// TIA Portal V15.1 export
// export: Created 2024-05-17T05:38:40.0003593Z, ExportSetting WithDefaults, DisplayName Totally Integrated Automation Portal, DisplayVersion V15.1 Update 5, DisplayName TIA Portal Openness, DisplayVersion V15.1 Update 5, DisplayName SINAMICS Startdrive Advanced, DisplayVersion V15.1, DisplayName G130, G150, S120, S150, SINAMICS MV, S210, DisplayVersion V15.1, DisplayName G110M, G120, G120C, G120D, G120P, DisplayVersion V15.1, DisplayName STEP 7 Professional, DisplayVersion V15.1 Update 5, DisplayName STEP 7 Safety, DisplayVersion V15.1, DisplayName WinCC Professional, DisplayVersion V15.1 Update 5, DisplayName SIMATIC Visualization Architect, DisplayVersion V15.1
FUNCTION_BLOCK "LGBProcessLighting"   // FB6697, FBD
TITLE = LGBProcessLighting
{ S7_Optimized_Access := 'TRUE' }
VERSION : 0.1
// stored: AutoNumber false, IsIECCheckEnabled false, IsRetainMemResEnabled false, MemoryReserve 100, SetENOAutomatically False, UDAEnableTagReadback false
   VAR_INPUT
      I_StartProduction { ExternalAccessible := 'False'; ExternalVisible := 'False'; ExternalWritable := 'False'} : Bool;   // Start Production line
      I_StopProduction { ExternalAccessible := 'False'; ExternalVisible := 'False'; ExternalWritable := 'False'} : Bool;   // Stop Production line
      I_StartReqCR { ExternalAccessible := 'False'; ExternalVisible := 'False'; ExternalWritable := 'False'} : Bool;   // Start request by controlroom
      I_StoppedByCR { ExternalAccessible := 'False'; ExternalVisible := 'False'; ExternalWritable := 'False'} : Bool;   // Production line stopped by control room
      I_BodyNumber { ExternalAccessible := 'False'; ExternalVisible := 'False'; ExternalWritable := 'False'} : DWord;   // Body number
      I_TopCoatColour { ExternalAccessible := 'False'; ExternalVisible := 'False'; ExternalWritable := 'False'} : Int;   // Top coat colour
      I_ColourGroup { ExternalAccessible := 'False'; ExternalVisible := 'False'; ExternalWritable := 'False'} : "ColourGroup";   // High speed value 0-100% / Colour Group
   END_VAR
   VAR_OUTPUT
      O_BreakMode { ExternalAccessible := 'False'; ExternalVisible := 'False'; ExternalWritable := 'False'} : Bool;   // Output 1 - Break Mode
      O_Intensity1 { ExternalAccessible := 'False'; ExternalVisible := 'False'; ExternalWritable := 'False'} : Bool;   // Output 2 - Intensity 1
      O_Intensity2 { ExternalAccessible := 'False'; ExternalVisible := 'False'; ExternalWritable := 'False'} : Bool;   // Output 3 - Intensity 2
      O_Intensity3 { ExternalAccessible := 'False'; ExternalVisible := 'False'; ExternalWritable := 'False'} : Bool;   // Output 4 - Intensity 3
      O_AlarmABCondition { ExternalAccessible := 'False'; ExternalVisible := 'False'; ExternalWritable := 'False'} : Bool;   // Alarm AB Condition
      O_AlarmA { ExternalAccessible := 'False'; ExternalVisible := 'False'; ExternalWritable := 'False'} : Bool;   // Alarm A
      O_AlarmB { ExternalAccessible := 'False'; ExternalVisible := 'False'; ExternalWritable := 'False'} : Bool;   // Alarm B
      O_AlarmC { ExternalAccessible := 'False'; ExternalVisible := 'False'; ExternalWritable := 'False'} : Bool;   // Alarm C
      O_AlarmD { ExternalAccessible := 'False'; ExternalVisible := 'False'; ExternalWritable := 'False'} : Bool;   // Alarm D
      H_AlarmDWord { ExternalAccessible := 'False'; ExternalVisible := 'False'; ExternalWritable := 'False'} : DWord;   // Alarm Word
   END_VAR
   VAR_IN_OUT
      H_HMI : "H_HMI";   // Icon Animation
      H_GBProcessLighting : "H_GBProcessLighting";   // Animation
      C_ProcessLightingConfig : "ProcessLightingConfig";   // Config
      IO_IDWorkStation { ExternalAccessible := 'False'; ExternalVisible := 'False'; ExternalWritable := 'False'} : Int;   // ID
      IO_GlobalOutput { ExternalAccessible := 'False'; ExternalVisible := 'False'; ExternalWritable := 'False'} : Bool;   // Global output
   END_VAR
   VAR
      AC_TopCoatColour { ExternalAccessible := 'False'; ExternalVisible := 'False'; ExternalWritable := 'False'} : Bool;   // Top Coat Colour is not configured in a colour group
      AD_ForceBreakMode { ExternalAccessible := 'False'; ExternalVisible := 'False'; ExternalWritable := 'False'} : Bool;   // Force process lighting active for Break Mode
      AD_ForceIntensity1 { ExternalAccessible := 'False'; ExternalVisible := 'False'; ExternalWritable := 'False'} : Bool;   // Force process lighting active for Intensity 1
      AD_ForceIntensity2 { ExternalAccessible := 'False'; ExternalVisible := 'False'; ExternalWritable := 'False'} : Bool;   // Force process lighting active for Intensity 2
      AD_ForceIntensity3 { ExternalAccessible := 'False'; ExternalVisible := 'False'; ExternalWritable := 'False'} : Bool;   // Force process lighting active for Intensity 3
      AlarmA { ExternalAccessible := 'False'; ExternalVisible := 'False'; ExternalWritable := 'False'} : Bool;   // Alarm A
      AlarmB { ExternalAccessible := 'False'; ExternalVisible := 'False'; ExternalWritable := 'False'} : Bool;   // Alarm B
      AlarmC { ExternalAccessible := 'False'; ExternalVisible := 'False'; ExternalWritable := 'False'} : Bool;   // Alarm C
      AlarmD { ExternalAccessible := 'False'; ExternalVisible := 'False'; ExternalWritable := 'False'} : Bool;   // Alarm D
      AlarmABCondition { ExternalAccessible := 'False'; ExternalVisible := 'False'; ExternalWritable := 'False'} : Bool;   // Alarm AB Condition
   END_VAR
   VAR RETAIN
      SwitchOFFLighting { ExternalAccessible := 'False'; ExternalVisible := 'False'; ExternalWritable := 'False'} : Bool;   // Switch OFF process lighting, END of production
      ReqBreakMode { ExternalAccessible := 'False'; ExternalVisible := 'False'; ExternalWritable := 'False'} : Bool;   // Request Break Mode
      ReqIntensity1 { ExternalAccessible := 'False'; ExternalVisible := 'False'; ExternalWritable := 'False'} : Bool;   // Request Intensity 1
      ReqIntensity2 { ExternalAccessible := 'False'; ExternalVisible := 'False'; ExternalWritable := 'False'} : Bool;   // Request Intensity 2
      ReqIntensity3 { ExternalAccessible := 'False'; ExternalVisible := 'False'; ExternalWritable := 'False'} : Bool;   // Request Intensity 3
      BreakMode { ExternalAccessible := 'False'; ExternalVisible := 'False'; ExternalWritable := 'False'} : Bool;   // Break Mode
      Intensity1 { ExternalAccessible := 'False'; ExternalVisible := 'False'; ExternalWritable := 'False'} : Bool;   // Intensity 1
      Intensity2 { ExternalAccessible := 'False'; ExternalVisible := 'False'; ExternalWritable := 'False'} : Bool;   // Intensity 2
      Intensity3 { ExternalAccessible := 'False'; ExternalVisible := 'False'; ExternalWritable := 'False'} : Bool;   // Intensity 3
   END_VAR
   VAR
      HMICmd_ForceBreakMode { ExternalAccessible := 'False'; ExternalVisible := 'False'; ExternalWritable := 'False'} : Bool;   // HMI Command - Force Break Mode
      HMICmd_ForceIntensity1 { ExternalAccessible := 'False'; ExternalVisible := 'False'; ExternalWritable := 'False'} : Bool;   // HMI Command - Force Intensity 1
      HMICmd_ForceIntensity2 { ExternalAccessible := 'False'; ExternalVisible := 'False'; ExternalWritable := 'False'} : Bool;   // HMI Command - Force Intensity 2
      HMICmd_ForceIntensity3 { ExternalAccessible := 'False'; ExternalVisible := 'False'; ExternalWritable := 'False'} : Bool;   // HMI Command - Force Intensity 3
      DelayBreakMode { ExternalAccessible := 'False'; ExternalVisible := 'False'; ExternalWritable := 'False'} : Bool;   // Delay Break Mode
      ActDelayTimeBreakMode { ExternalAccessible := 'False'; ExternalVisible := 'False'; ExternalWritable := 'False'} : Time;   // Actual delay time break mode
      IDWorkStation { ExternalAccessible := 'False'; ExternalVisible := 'False'; ExternalWritable := 'False'} : Bool;   // ID Workstation
      TopCoatColourLong { ExternalAccessible := 'False'; ExternalVisible := 'False'; ExternalWritable := 'False'} : Int;   // Top coat colour
      TopCoatColour { ExternalAccessible := 'False'; ExternalVisible := 'False'; ExternalWritable := 'False'} : Int;   // Top coat colour
      ColourGroup { ExternalAccessible := 'False'; ExternalVisible := 'False'; ExternalWritable := 'False'} : Int;   // Colour Group
      T_DelayBreakMode { ExternalAccessible := 'False'; ExternalVisible := 'False'; ExternalWritable := 'False'} : "LTimer";   // FB
      T_IDWorkStation { ExternalAccessible := 'False'; ExternalVisible := 'False'; ExternalWritable := 'False'} : "LTimer";   // FB
      _ColourGroup { ExternalAccessible := 'False'; ExternalVisible := 'False'; ExternalWritable := 'False'} : "LGBColourGroup";   // FB
   END_VAR
BEGIN

REGION Network 1: **** 1 - Inputs **** Extract HMI Commands
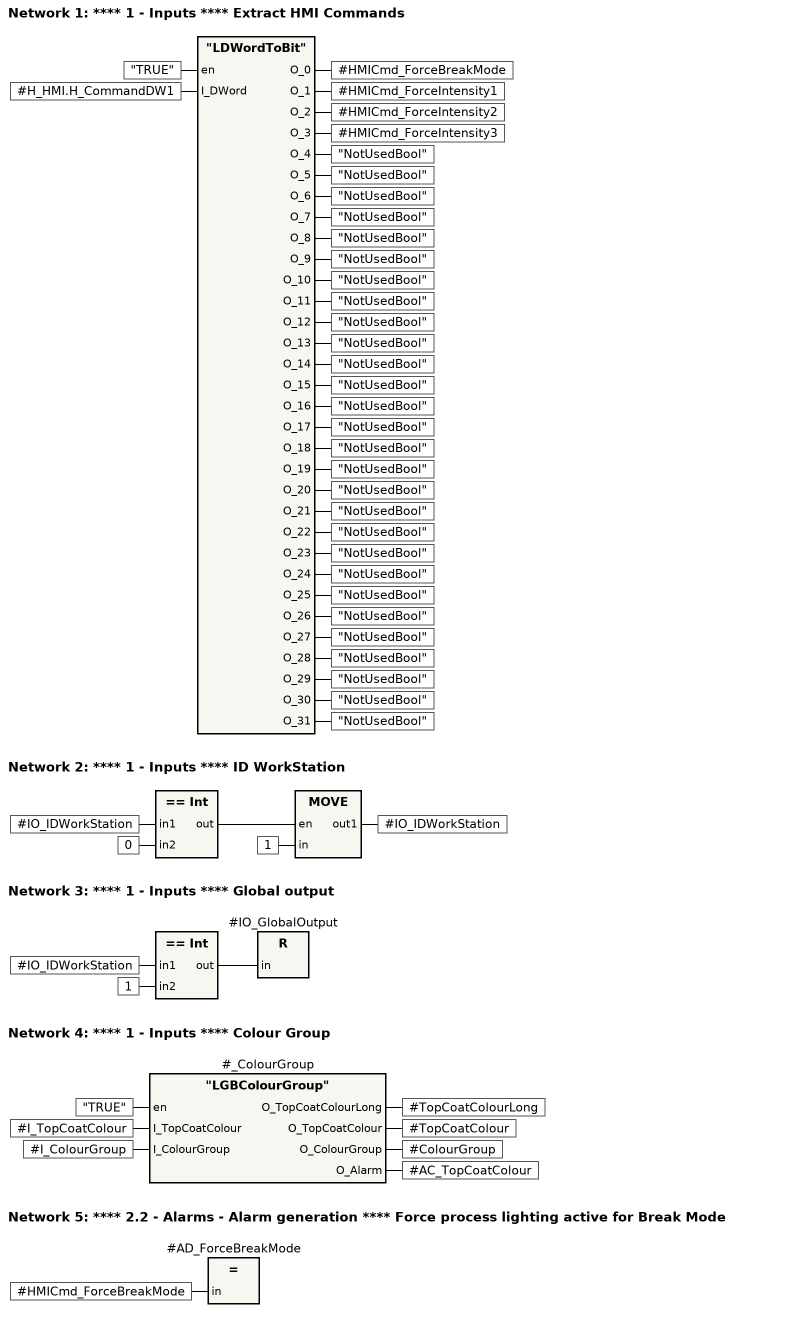
   IF "TRUE" THEN
       "LDWordToBit"(I_DWord := #H_HMI.H_CommandDW1,
                     O_0 => #HMICmd_ForceBreakMode,
                     O_1 => #HMICmd_ForceIntensity1,
                     O_2 => #HMICmd_ForceIntensity2,
                     O_3 => #HMICmd_ForceIntensity3,
                     O_4 => "NotUsedBool",
                     O_5 => "NotUsedBool",
                     O_6 => "NotUsedBool",
                     O_7 => "NotUsedBool",
                     O_8 => "NotUsedBool",
                     O_9 => "NotUsedBool",
                     O_10 => "NotUsedBool",
                     O_11 => "NotUsedBool",
                     O_12 => "NotUsedBool",
                     O_13 => "NotUsedBool",
                     O_14 => "NotUsedBool",
                     O_15 => "NotUsedBool",
                     O_16 => "NotUsedBool",
                     O_17 => "NotUsedBool",
                     O_18 => "NotUsedBool",
                     O_19 => "NotUsedBool",
                     O_20 => "NotUsedBool",
                     O_21 => "NotUsedBool",
                     O_22 => "NotUsedBool",
                     O_23 => "NotUsedBool",
                     O_24 => "NotUsedBool",
                     O_25 => "NotUsedBool",
                     O_26 => "NotUsedBool",
                     O_27 => "NotUsedBool",
                     O_28 => "NotUsedBool",
                     O_29 => "NotUsedBool",
                     O_30 => "NotUsedBool",
                     O_31 => "NotUsedBool");
   END_IF;
END_REGION

REGION Network 2: **** 1 - Inputs **** ID WorkStation
   IF #IO_IDWorkStation = 0 THEN #IO_IDWorkStation := 1; END_IF;
END_REGION

REGION Network 3: **** 1 - Inputs **** Global output
   IF #IO_IDWorkStation = 1 THEN #IO_GlobalOutput := FALSE; END_IF;
END_REGION

REGION Network 4: **** 1 - Inputs **** Colour Group
   IF "TRUE" THEN
       #_ColourGroup(I_TopCoatColour := #I_TopCoatColour,   // "LGBColourGroup"
                     I_ColourGroup := #I_ColourGroup,
                     O_TopCoatColourLong => #TopCoatColourLong,
                     O_TopCoatColour => #TopCoatColour,
                     O_ColourGroup => #ColourGroup,
                     O_Alarm => #AC_TopCoatColour);
   END_IF;
END_REGION

REGION Network 5: **** 2.2 - Alarms - Alarm generation **** Force process lighting active for Break Mode
   #AD_ForceBreakMode := #HMICmd_ForceBreakMode;
END_REGION

REGION Network 6: **** 2.2 - Alarms - Alarm generation **** Force process lighting active for Intensity 1
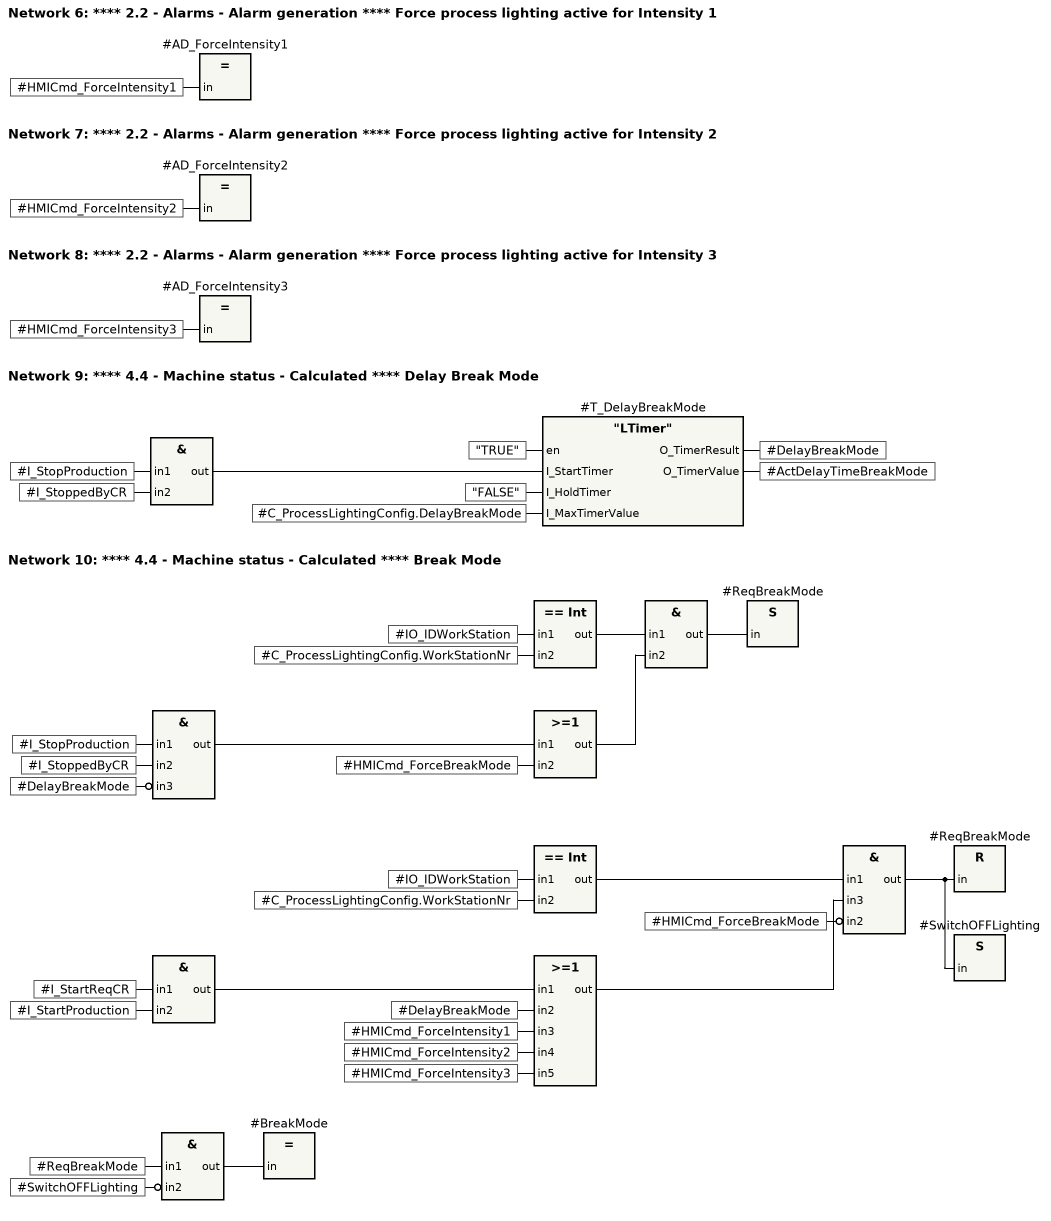
   #AD_ForceIntensity1 := #HMICmd_ForceIntensity1;
END_REGION

REGION Network 7: **** 2.2 - Alarms - Alarm generation **** Force process lighting active for Intensity 2
   #AD_ForceIntensity2 := #HMICmd_ForceIntensity2;
END_REGION

REGION Network 8: **** 2.2 - Alarms - Alarm generation **** Force process lighting active for Intensity 3
   #AD_ForceIntensity3 := #HMICmd_ForceIntensity3;
END_REGION

REGION Network 9: **** 4.4 - Machine status - Calculated **** Delay Break Mode
   IF "TRUE" THEN
       #T_DelayBreakMode(I_StartTimer := #I_StopProduction AND #I_StoppedByCR,   // "LTimer"
                         I_HoldTimer := "FALSE",
                         I_MaxTimerValue := #C_ProcessLightingConfig.DelayBreakMode,
                         O_TimerResult => #DelayBreakMode,
                         O_TimerValue => #ActDelayTimeBreakMode);
   END_IF;
END_REGION

REGION Network 10: **** 4.4 - Machine status - Calculated **** Break Mode
   IF (#IO_IDWorkStation = #C_ProcessLightingConfig.WorkStationNr) AND ((#I_StopProduction AND #I_StoppedByCR AND NOT #DelayBreakMode) OR #HMICmd_ForceBreakMode) THEN
       #ReqBreakMode := TRUE;
   END_IF;
   IF (#IO_IDWorkStation = #C_ProcessLightingConfig.WorkStationNr) AND ((#I_StartReqCR AND #I_StartProduction) OR #DelayBreakMode OR #HMICmd_ForceIntensity1 OR #HMICmd_ForceIntensity2 OR #HMICmd_ForceIntensity3) AND NOT #HMICmd_ForceBreakMode THEN
       #ReqBreakMode := FALSE;
       #SwitchOFFLighting := TRUE;
   END_IF;
   #BreakMode := #ReqBreakMode AND NOT #SwitchOFFLighting;
END_REGION

REGION Network 11: **** 4.4 - Machine status - Calculated **** Switch OFF process lighting, END of production
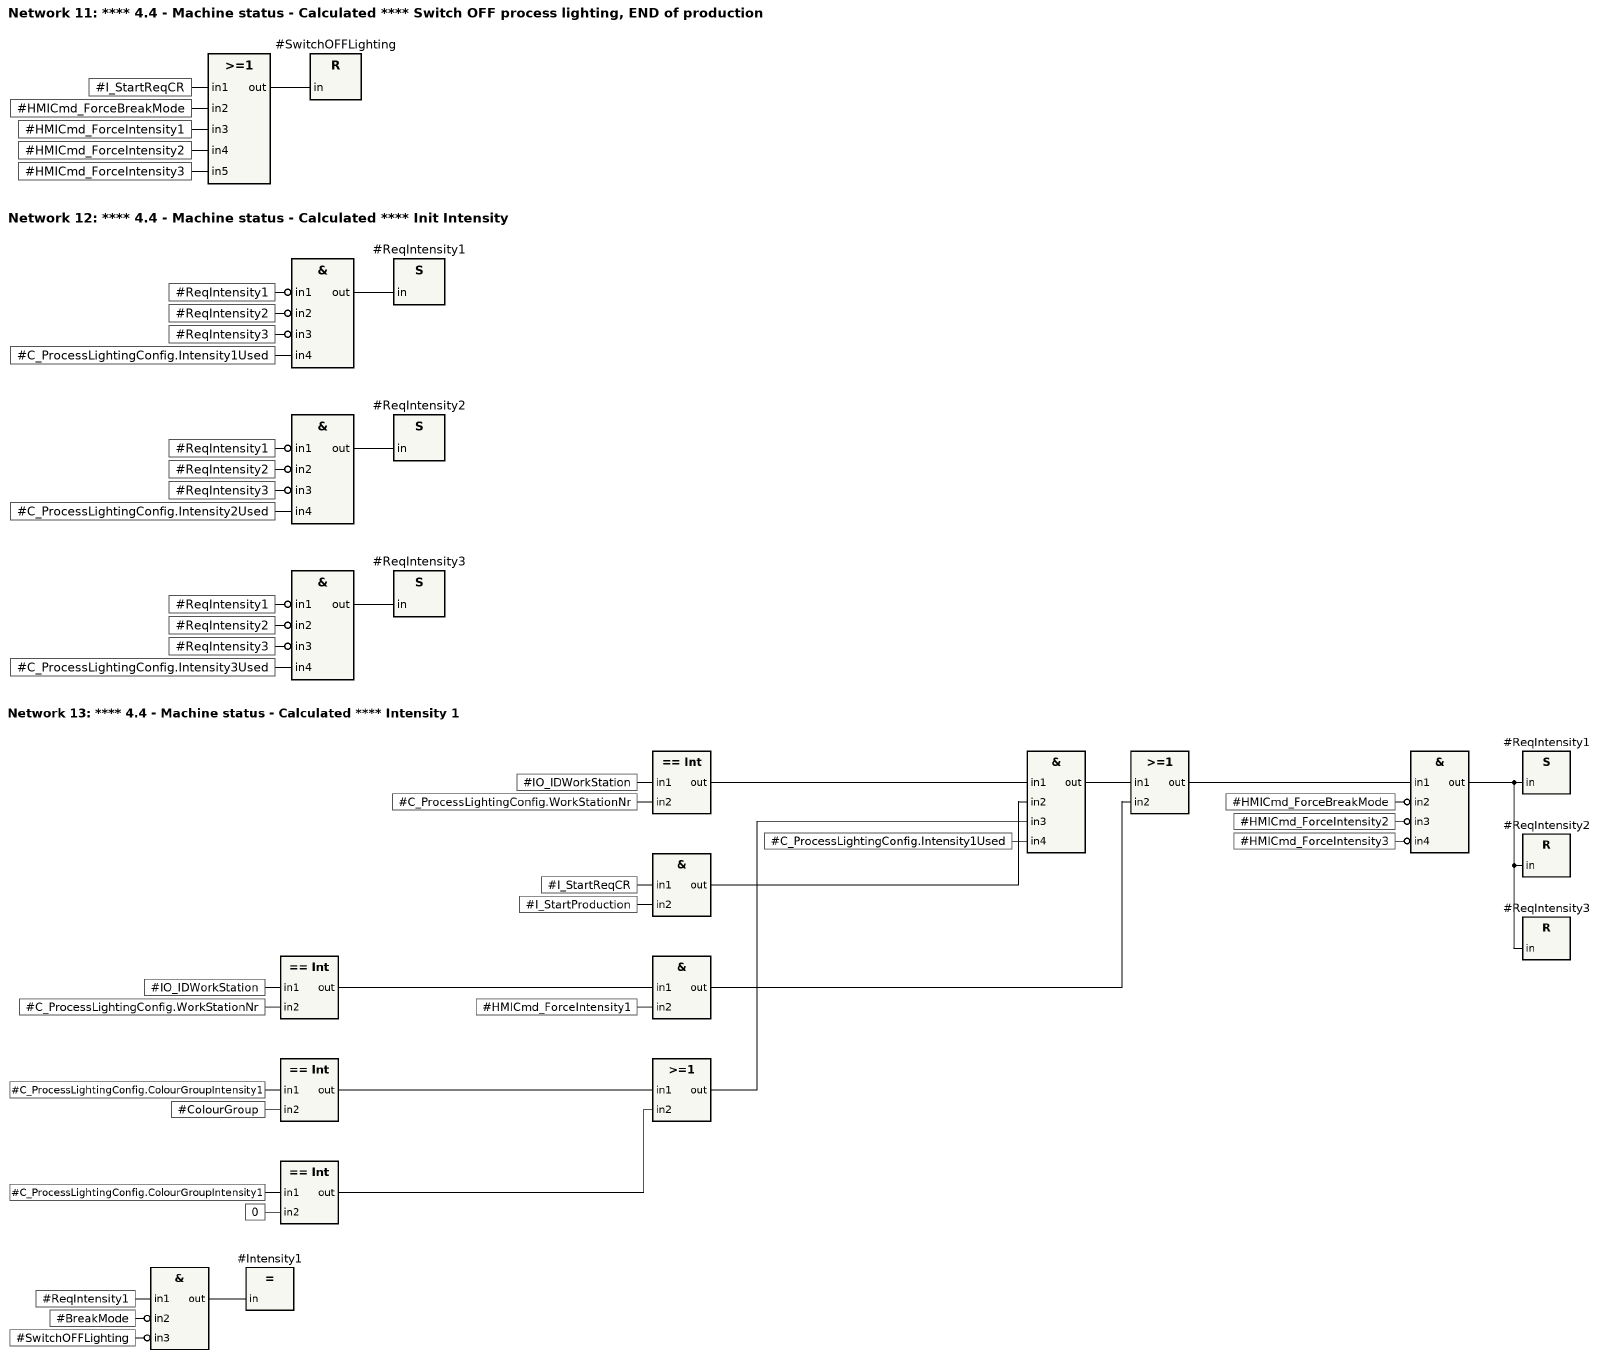
   IF #I_StartReqCR OR #HMICmd_ForceBreakMode OR #HMICmd_ForceIntensity1 OR #HMICmd_ForceIntensity2 OR #HMICmd_ForceIntensity3 THEN
       #SwitchOFFLighting := FALSE;
   END_IF;
END_REGION

REGION Network 12: **** 4.4 - Machine status - Calculated **** Init Intensity
   IF NOT #ReqIntensity1 AND NOT #ReqIntensity2 AND NOT #ReqIntensity3 AND #C_ProcessLightingConfig.Intensity1Used THEN
       #ReqIntensity1 := TRUE;
   END_IF;
   IF NOT #ReqIntensity1 AND NOT #ReqIntensity2 AND NOT #ReqIntensity3 AND #C_ProcessLightingConfig.Intensity2Used THEN
       #ReqIntensity2 := TRUE;
   END_IF;
   IF NOT #ReqIntensity1 AND NOT #ReqIntensity2 AND NOT #ReqIntensity3 AND #C_ProcessLightingConfig.Intensity3Used THEN
       #ReqIntensity3 := TRUE;
   END_IF;
END_REGION

REGION Network 13: **** 4.4 - Machine status - Calculated **** Intensity 1
   IF (((#IO_IDWorkStation = #C_ProcessLightingConfig.WorkStationNr) AND #I_StartReqCR AND #I_StartProduction AND ((#C_ProcessLightingConfig.ColourGroupIntensity1 = #ColourGroup) OR (#C_ProcessLightingConfig.ColourGroupIntensity1 = 0)) AND #C_ProcessLightingConfig.Intensity1Used) OR ((#IO_IDWorkStation = #C_ProcessLightingConfig.WorkStationNr) AND #HMICmd_ForceIntensity1)) AND NOT #HMICmd_ForceBreakMode AND NOT #HMICmd_ForceIntensity2 AND NOT #HMICmd_ForceIntensity3 THEN
       #ReqIntensity1 := TRUE;
       #ReqIntensity2 := FALSE;
       #ReqIntensity3 := FALSE;
   END_IF;
   #Intensity1 := #ReqIntensity1 AND NOT #BreakMode AND NOT #SwitchOFFLighting;
END_REGION

REGION Network 14: **** 4.4 - Machine status - Calculated **** Intensity 2
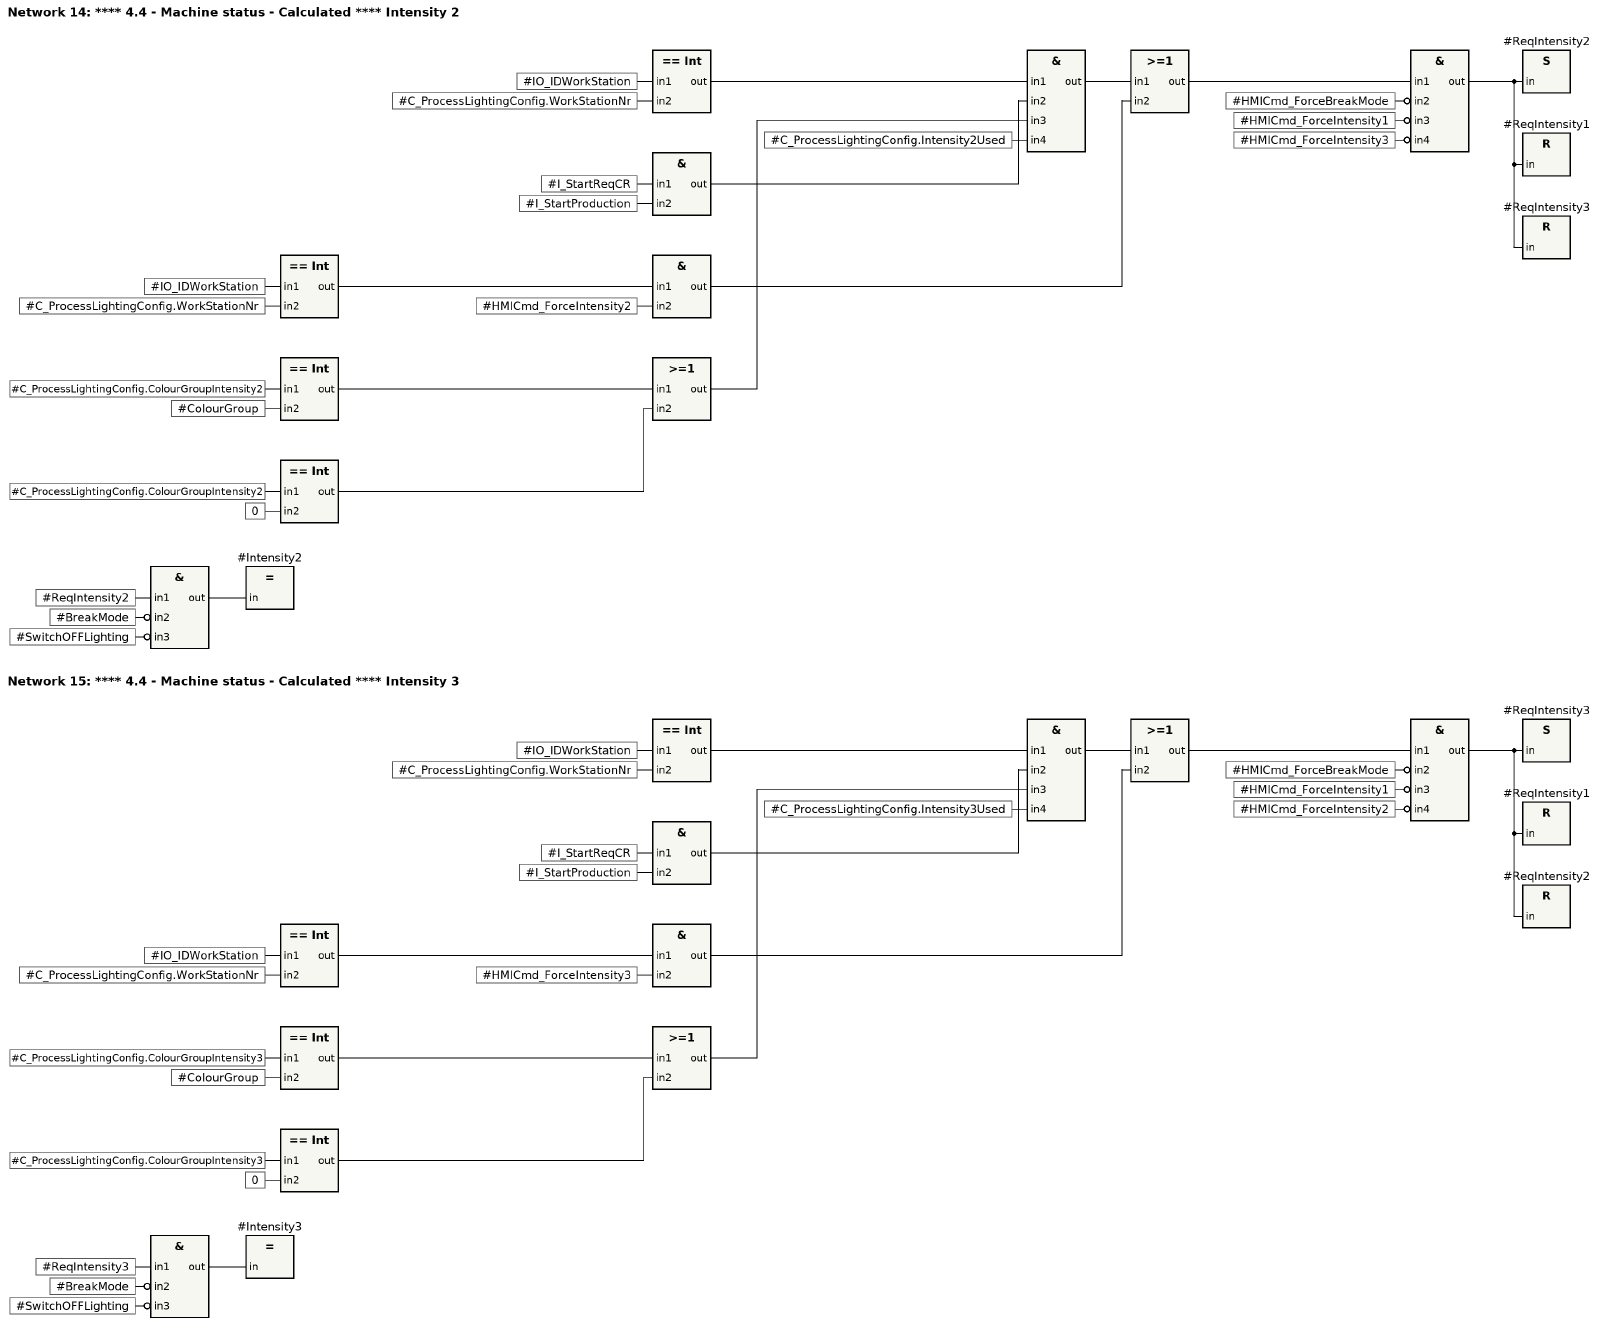
   IF (((#IO_IDWorkStation = #C_ProcessLightingConfig.WorkStationNr) AND #I_StartReqCR AND #I_StartProduction AND ((#C_ProcessLightingConfig.ColourGroupIntensity2 = #ColourGroup) OR (#C_ProcessLightingConfig.ColourGroupIntensity2 = 0)) AND #C_ProcessLightingConfig.Intensity2Used) OR ((#IO_IDWorkStation = #C_ProcessLightingConfig.WorkStationNr) AND #HMICmd_ForceIntensity2)) AND NOT #HMICmd_ForceBreakMode AND NOT #HMICmd_ForceIntensity1 AND NOT #HMICmd_ForceIntensity3 THEN
       #ReqIntensity2 := TRUE;
       #ReqIntensity1 := FALSE;
       #ReqIntensity3 := FALSE;
   END_IF;
   #Intensity2 := #ReqIntensity2 AND NOT #BreakMode AND NOT #SwitchOFFLighting;
END_REGION

REGION Network 15: **** 4.4 - Machine status - Calculated **** Intensity 3
   IF (((#IO_IDWorkStation = #C_ProcessLightingConfig.WorkStationNr) AND #I_StartReqCR AND #I_StartProduction AND ((#C_ProcessLightingConfig.ColourGroupIntensity3 = #ColourGroup) OR (#C_ProcessLightingConfig.ColourGroupIntensity3 = 0)) AND #C_ProcessLightingConfig.Intensity3Used) OR ((#IO_IDWorkStation = #C_ProcessLightingConfig.WorkStationNr) AND #HMICmd_ForceIntensity3)) AND NOT #HMICmd_ForceBreakMode AND NOT #HMICmd_ForceIntensity1 AND NOT #HMICmd_ForceIntensity2 THEN
       #ReqIntensity3 := TRUE;
       #ReqIntensity1 := FALSE;
       #ReqIntensity2 := FALSE;
   END_IF;
   #Intensity3 := #ReqIntensity3 AND NOT #BreakMode AND NOT #SwitchOFFLighting;
END_REGION

REGION Network 16: **** 4.4 - Machine status - Calculated **** ID WorkStation
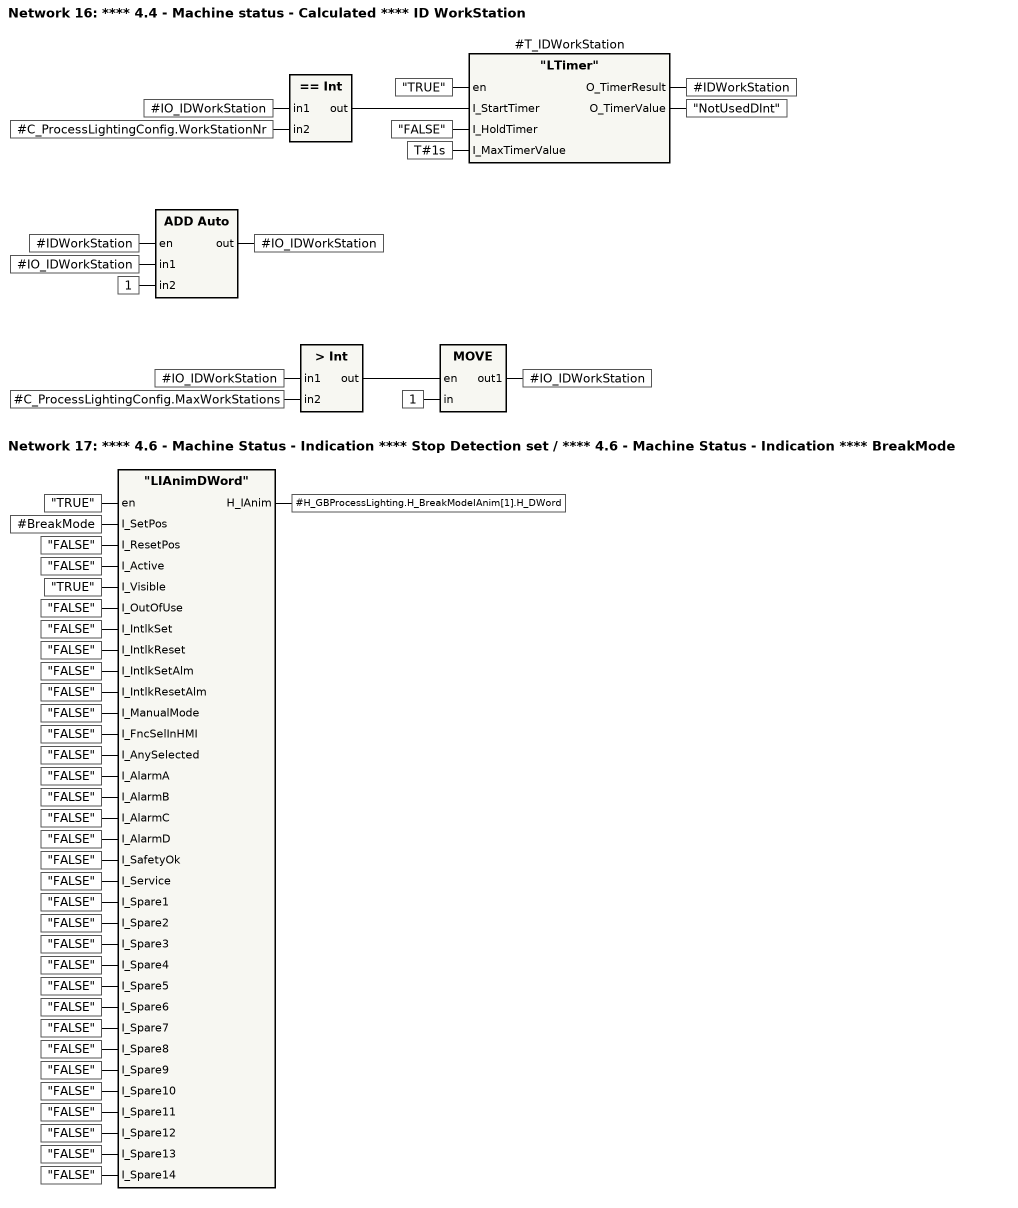
   IF "TRUE" THEN
       #T_IDWorkStation(I_StartTimer := #IO_IDWorkStation = #C_ProcessLightingConfig.WorkStationNr,   // "LTimer"
                        I_HoldTimer := "FALSE",
                        I_MaxTimerValue := T#1s,
                        O_TimerResult => #IDWorkStation,
                        O_TimerValue => "NotUsedDInt");
   END_IF;
   IF #IDWorkStation THEN #IO_IDWorkStation := #IO_IDWorkStation + 1; END_IF;
   IF #IO_IDWorkStation > #C_ProcessLightingConfig.MaxWorkStations THEN #IO_IDWorkStation := 1; END_IF;
END_REGION

REGION Network 17: **** 4.6 - Machine Status - Indication **** Stop Detection set / **** 4.6 - Machine Status - Indication **** BreakMode
   // Stop Detection set
   IF "TRUE" THEN
       "LIAnimDWord"(I_SetPos := #BreakMode,
                     I_ResetPos := "FALSE",
                     I_Active := "FALSE",
                     I_Visible := "TRUE",
                     I_OutOfUse := "FALSE",
                     I_IntlkSet := "FALSE",
                     I_IntlkReset := "FALSE",
                     I_IntlkSetAlm := "FALSE",
                     I_IntlkResetAlm := "FALSE",
                     I_ManualMode := "FALSE",
                     I_FncSelInHMI := "FALSE",
                     I_AnySelected := "FALSE",
                     I_AlarmA := "FALSE",
                     I_AlarmB := "FALSE",
                     I_AlarmC := "FALSE",
                     I_AlarmD := "FALSE",
                     I_SafetyOk := "FALSE",
                     I_Service := "FALSE",
                     I_Spare1 := "FALSE",
                     I_Spare2 := "FALSE",
                     I_Spare3 := "FALSE",
                     I_Spare4 := "FALSE",
                     I_Spare5 := "FALSE",
                     I_Spare6 := "FALSE",
                     I_Spare7 := "FALSE",
                     I_Spare8 := "FALSE",
                     I_Spare9 := "FALSE",
                     I_Spare10 := "FALSE",
                     I_Spare11 := "FALSE",
                     I_Spare12 := "FALSE",
                     I_Spare13 := "FALSE",
                     I_Spare14 := "FALSE",
                     H_IAnim => #H_GBProcessLighting.H_BreakModeIAnim[1].H_DWord);
   END_IF;
END_REGION

REGION Network 18: **** 4.6 - Machine Status - Indication **** Stop Detection set / **** 4.6 - Machine Status - Indication **** Intensity1
   // Stop Detection set
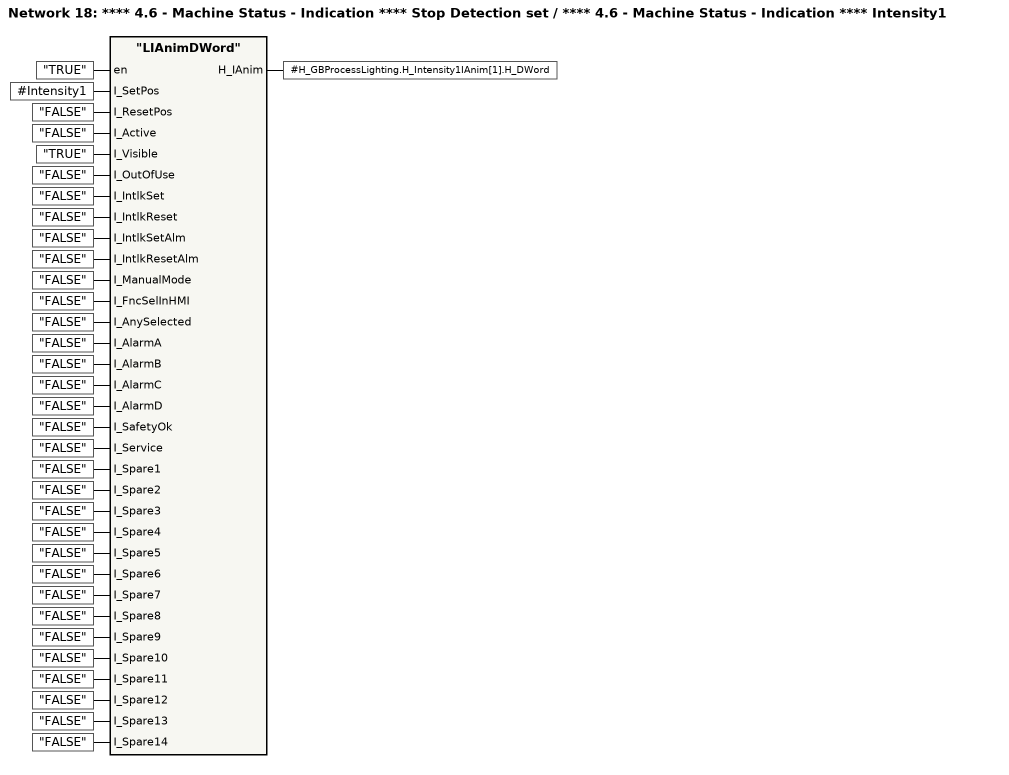
   IF "TRUE" THEN
       "LIAnimDWord"(I_SetPos := #Intensity1,
                     I_ResetPos := "FALSE",
                     I_Active := "FALSE",
                     I_Visible := "TRUE",
                     I_OutOfUse := "FALSE",
                     I_IntlkSet := "FALSE",
                     I_IntlkReset := "FALSE",
                     I_IntlkSetAlm := "FALSE",
                     I_IntlkResetAlm := "FALSE",
                     I_ManualMode := "FALSE",
                     I_FncSelInHMI := "FALSE",
                     I_AnySelected := "FALSE",
                     I_AlarmA := "FALSE",
                     I_AlarmB := "FALSE",
                     I_AlarmC := "FALSE",
                     I_AlarmD := "FALSE",
                     I_SafetyOk := "FALSE",
                     I_Service := "FALSE",
                     I_Spare1 := "FALSE",
                     I_Spare2 := "FALSE",
                     I_Spare3 := "FALSE",
                     I_Spare4 := "FALSE",
                     I_Spare5 := "FALSE",
                     I_Spare6 := "FALSE",
                     I_Spare7 := "FALSE",
                     I_Spare8 := "FALSE",
                     I_Spare9 := "FALSE",
                     I_Spare10 := "FALSE",
                     I_Spare11 := "FALSE",
                     I_Spare12 := "FALSE",
                     I_Spare13 := "FALSE",
                     I_Spare14 := "FALSE",
                     H_IAnim => #H_GBProcessLighting.H_Intensity1IAnim[1].H_DWord);
   END_IF;
END_REGION

REGION Network 19: **** 4.6 - Machine Status - Indication **** Stop Detection set / **** 4.6 - Machine Status - Indication **** Intensity2
   // Stop Detection set
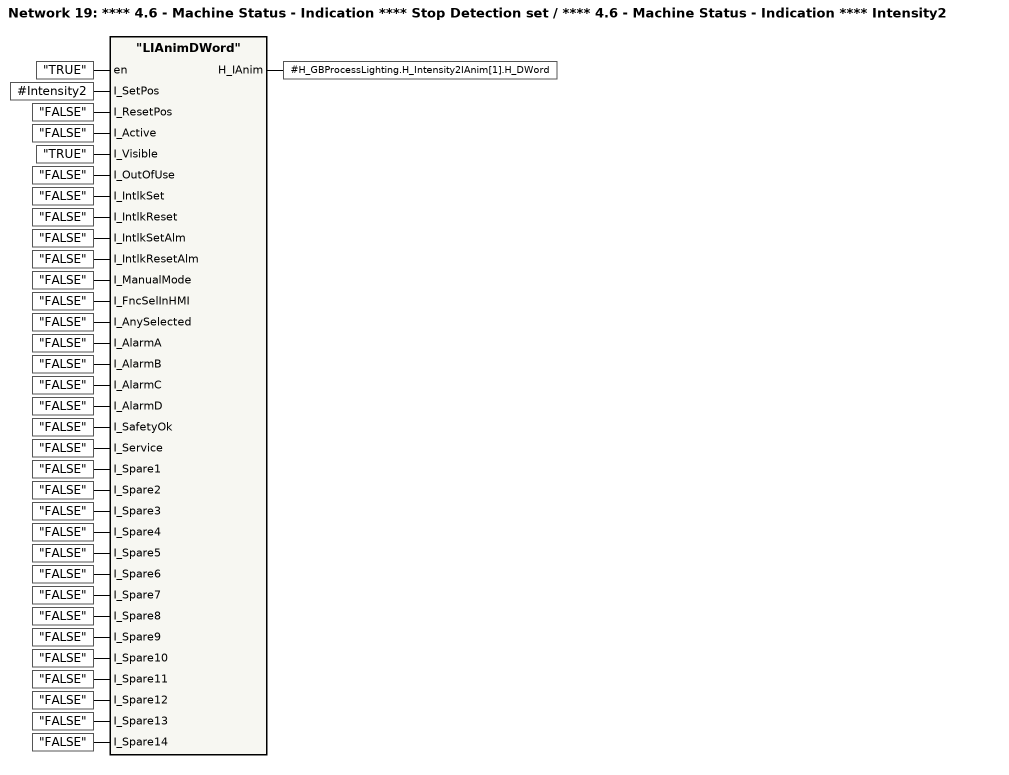
   IF "TRUE" THEN
       "LIAnimDWord"(I_SetPos := #Intensity2,
                     I_ResetPos := "FALSE",
                     I_Active := "FALSE",
                     I_Visible := "TRUE",
                     I_OutOfUse := "FALSE",
                     I_IntlkSet := "FALSE",
                     I_IntlkReset := "FALSE",
                     I_IntlkSetAlm := "FALSE",
                     I_IntlkResetAlm := "FALSE",
                     I_ManualMode := "FALSE",
                     I_FncSelInHMI := "FALSE",
                     I_AnySelected := "FALSE",
                     I_AlarmA := "FALSE",
                     I_AlarmB := "FALSE",
                     I_AlarmC := "FALSE",
                     I_AlarmD := "FALSE",
                     I_SafetyOk := "FALSE",
                     I_Service := "FALSE",
                     I_Spare1 := "FALSE",
                     I_Spare2 := "FALSE",
                     I_Spare3 := "FALSE",
                     I_Spare4 := "FALSE",
                     I_Spare5 := "FALSE",
                     I_Spare6 := "FALSE",
                     I_Spare7 := "FALSE",
                     I_Spare8 := "FALSE",
                     I_Spare9 := "FALSE",
                     I_Spare10 := "FALSE",
                     I_Spare11 := "FALSE",
                     I_Spare12 := "FALSE",
                     I_Spare13 := "FALSE",
                     I_Spare14 := "FALSE",
                     H_IAnim => #H_GBProcessLighting.H_Intensity2IAnim[1].H_DWord);
   END_IF;
END_REGION

REGION Network 20: **** 4.6 - Machine Status - Indication **** Stop Detection set / **** 4.6 - Machine Status - Indication **** Intensity3
   // Stop Detection set
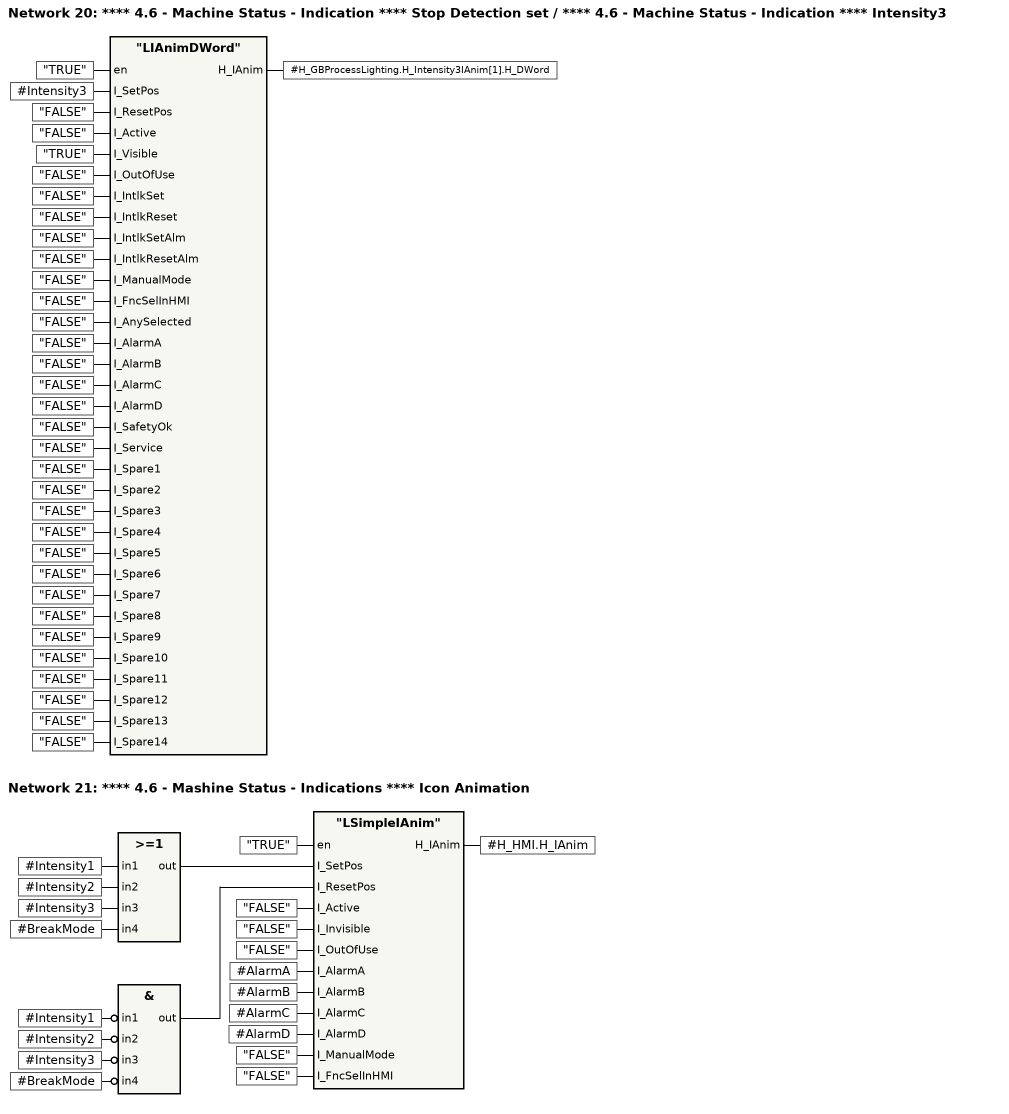
   IF "TRUE" THEN
       "LIAnimDWord"(I_SetPos := #Intensity3,
                     I_ResetPos := "FALSE",
                     I_Active := "FALSE",
                     I_Visible := "TRUE",
                     I_OutOfUse := "FALSE",
                     I_IntlkSet := "FALSE",
                     I_IntlkReset := "FALSE",
                     I_IntlkSetAlm := "FALSE",
                     I_IntlkResetAlm := "FALSE",
                     I_ManualMode := "FALSE",
                     I_FncSelInHMI := "FALSE",
                     I_AnySelected := "FALSE",
                     I_AlarmA := "FALSE",
                     I_AlarmB := "FALSE",
                     I_AlarmC := "FALSE",
                     I_AlarmD := "FALSE",
                     I_SafetyOk := "FALSE",
                     I_Service := "FALSE",
                     I_Spare1 := "FALSE",
                     I_Spare2 := "FALSE",
                     I_Spare3 := "FALSE",
                     I_Spare4 := "FALSE",
                     I_Spare5 := "FALSE",
                     I_Spare6 := "FALSE",
                     I_Spare7 := "FALSE",
                     I_Spare8 := "FALSE",
                     I_Spare9 := "FALSE",
                     I_Spare10 := "FALSE",
                     I_Spare11 := "FALSE",
                     I_Spare12 := "FALSE",
                     I_Spare13 := "FALSE",
                     I_Spare14 := "FALSE",
                     H_IAnim => #H_GBProcessLighting.H_Intensity3IAnim[1].H_DWord);
   END_IF;
END_REGION

REGION Network 21: **** 4.6 - Mashine Status - Indications **** Icon Animation
   // Icon Animation
   IF "TRUE" THEN
       "LSimpleIAnim"(I_SetPos := #Intensity1 OR #Intensity2 OR #Intensity3 OR #BreakMode,
                      I_ResetPos := NOT #Intensity1 AND NOT #Intensity2 AND NOT #Intensity3 AND NOT #BreakMode,
                      I_Active := "FALSE",
                      I_Invisible := "FALSE",
                      I_OutOfUse := "FALSE",
                      I_AlarmA := #AlarmA,
                      I_AlarmB := #AlarmB,
                      I_AlarmC := #AlarmC,
                      I_AlarmD := #AlarmD,
                      I_ManualMode := "FALSE",
                      I_FncSelInHMI := "FALSE",
                      H_IAnim => #H_HMI.H_IAnim);
   END_IF;
END_REGION

REGION Network 22: **** 4.6 - Machine status - Indications **** Icon Animation2
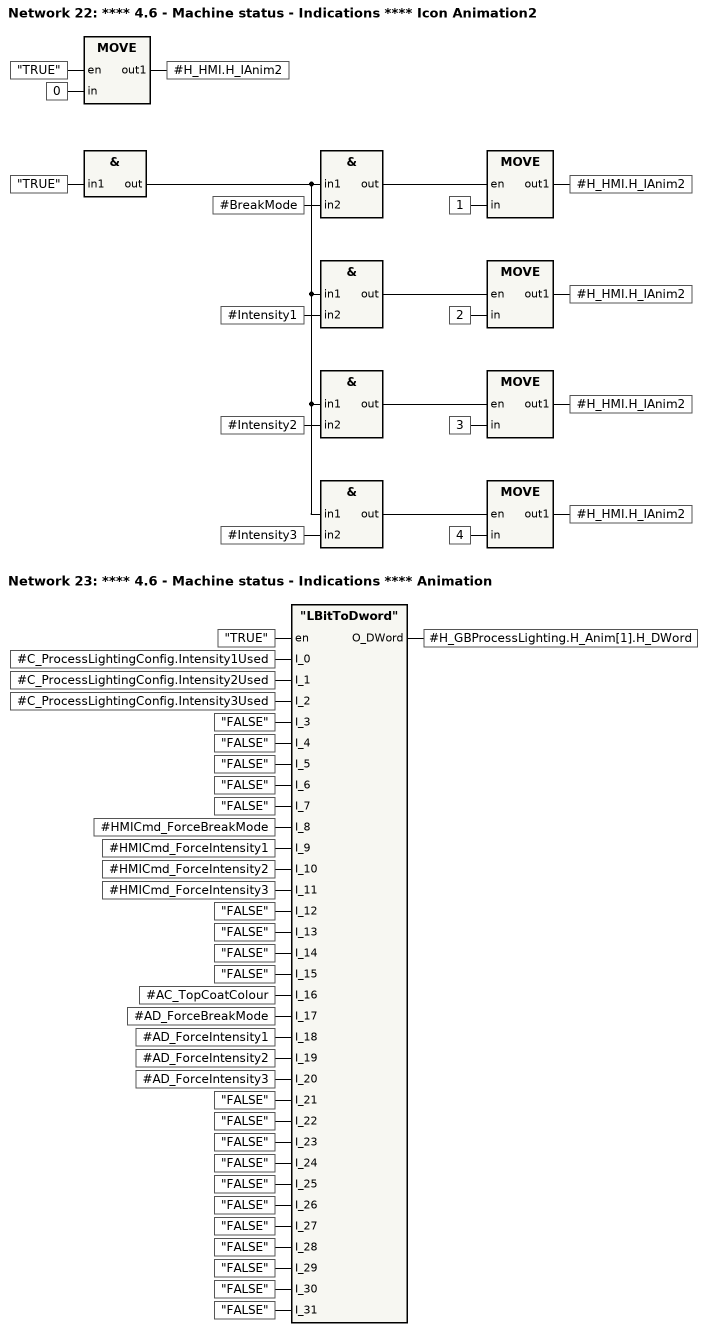
   IF "TRUE" THEN #H_HMI.H_IAnim2 := 0; END_IF;
   IF "TRUE" AND #BreakMode THEN #H_HMI.H_IAnim2 := 1; END_IF;
   IF "TRUE" AND #Intensity1 THEN #H_HMI.H_IAnim2 := 2; END_IF;
   IF "TRUE" AND #Intensity2 THEN #H_HMI.H_IAnim2 := 3; END_IF;
   IF "TRUE" AND #Intensity3 THEN #H_HMI.H_IAnim2 := 4; END_IF;
END_REGION

REGION Network 23: **** 4.6 - Machine status - Indications **** Animation
   // Animation Word 1
   IF "TRUE" THEN
       "LBitToDword"(I_0 := #C_ProcessLightingConfig.Intensity1Used,
                     I_1 := #C_ProcessLightingConfig.Intensity2Used,
                     I_2 := #C_ProcessLightingConfig.Intensity3Used,
                     I_3 := "FALSE",
                     I_4 := "FALSE",
                     I_5 := "FALSE",
                     I_6 := "FALSE",
                     I_7 := "FALSE",
                     I_8 := #HMICmd_ForceBreakMode,
                     I_9 := #HMICmd_ForceIntensity1,
                     I_10 := #HMICmd_ForceIntensity2,
                     I_11 := #HMICmd_ForceIntensity3,
                     I_12 := "FALSE",
                     I_13 := "FALSE",
                     I_14 := "FALSE",
                     I_15 := "FALSE",
                     I_16 := #AC_TopCoatColour,
                     I_17 := #AD_ForceBreakMode,
                     I_18 := #AD_ForceIntensity1,
                     I_19 := #AD_ForceIntensity2,
                     I_20 := #AD_ForceIntensity3,
                     I_21 := "FALSE",
                     I_22 := "FALSE",
                     I_23 := "FALSE",
                     I_24 := "FALSE",
                     I_25 := "FALSE",
                     I_26 := "FALSE",
                     I_27 := "FALSE",
                     I_28 := "FALSE",
                     I_29 := "FALSE",
                     I_30 := "FALSE",
                     I_31 := "FALSE",
                     O_DWord => #H_GBProcessLighting.H_Anim[1].H_DWord);
   END_IF;
END_REGION

REGION Network 24: **** 4.6 - Machine status - Indications **** Animation
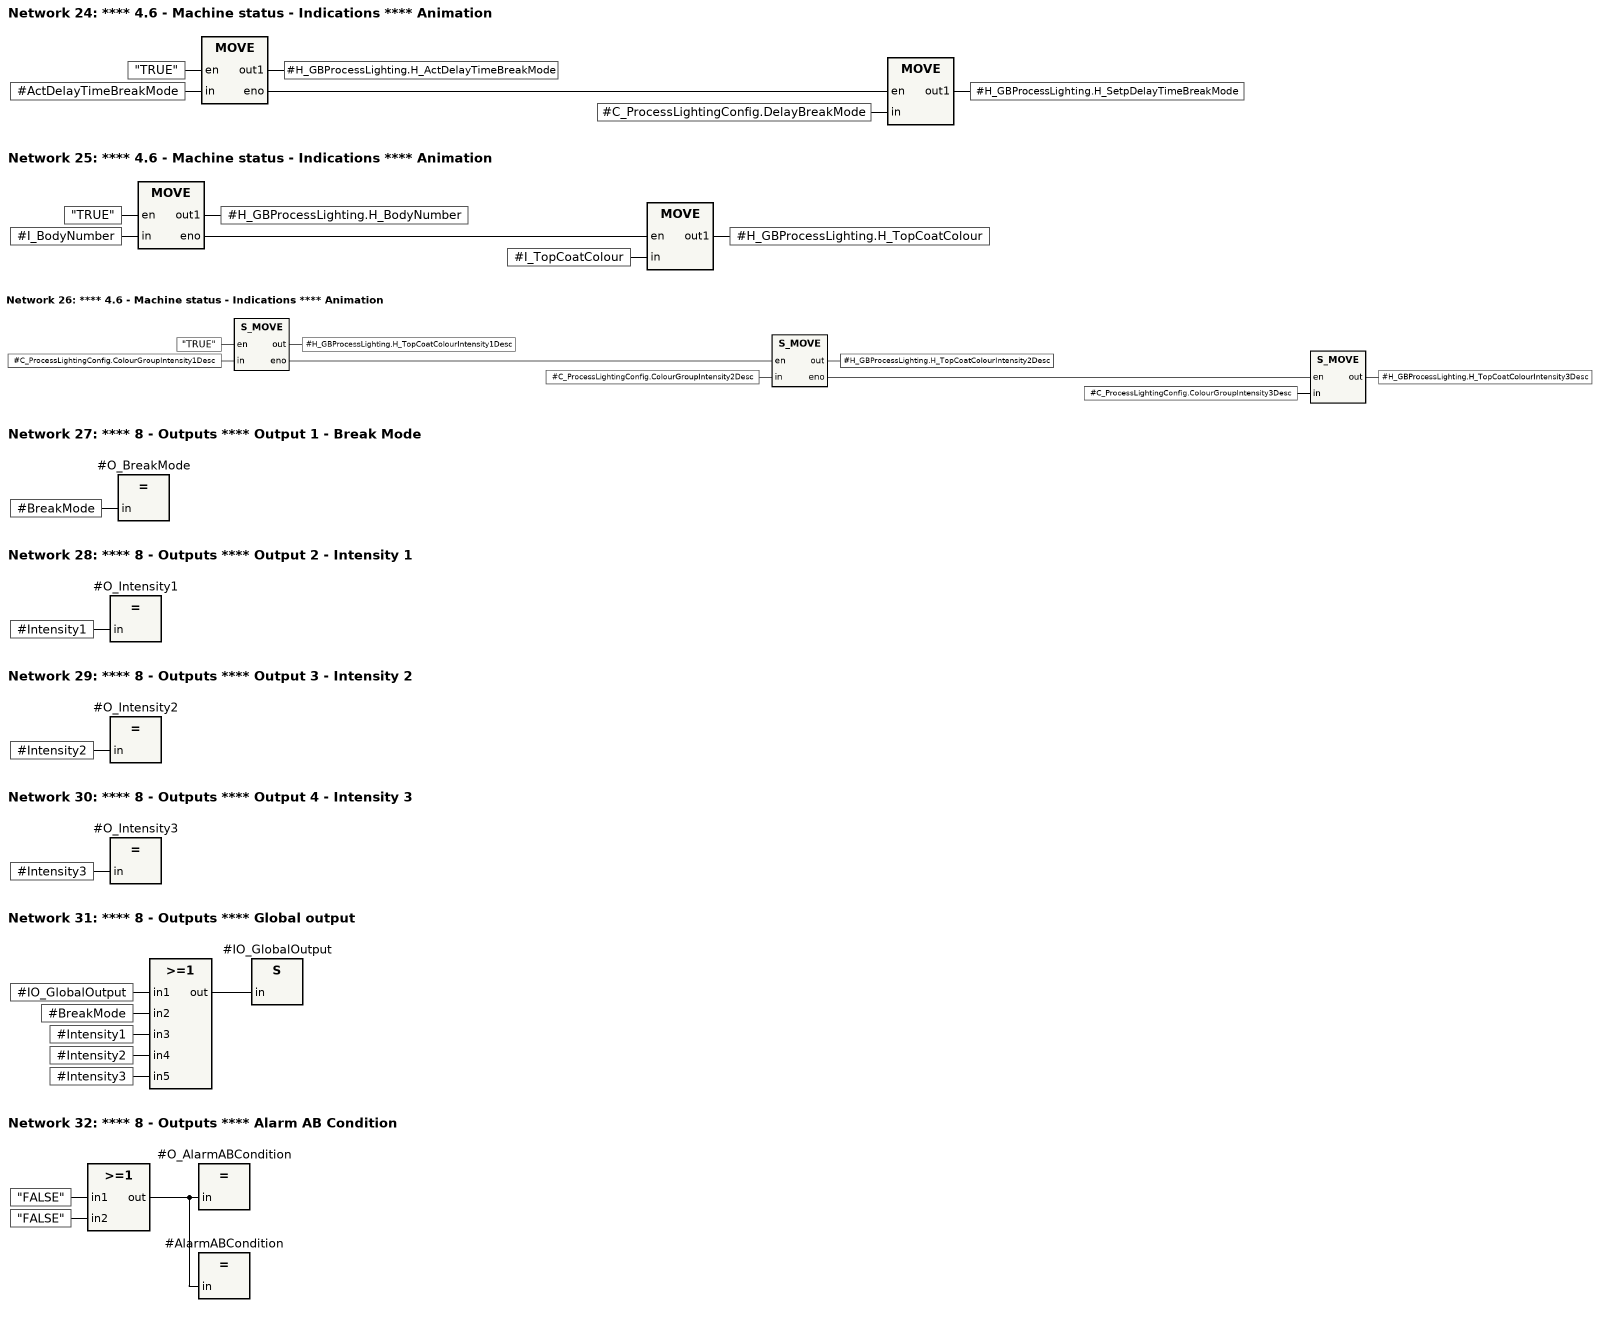
   IF "TRUE" THEN
       #H_GBProcessLighting.H_ActDelayTimeBreakMode := #ActDelayTimeBreakMode;
       #H_GBProcessLighting.H_SetpDelayTimeBreakMode := #C_ProcessLightingConfig.DelayBreakMode;
   END_IF;
END_REGION

REGION Network 25: **** 4.6 - Machine status - Indications **** Animation
   IF "TRUE" THEN
       #H_GBProcessLighting.H_BodyNumber := #I_BodyNumber;
       #H_GBProcessLighting.H_TopCoatColour := #I_TopCoatColour;
   END_IF;
END_REGION

REGION Network 26: **** 4.6 - Machine status - Indications **** Animation
   IF "TRUE" THEN
       #H_GBProcessLighting.H_TopCoatColourIntensity1Desc := #C_ProcessLightingConfig.ColourGroupIntensity1Desc;
       #H_GBProcessLighting.H_TopCoatColourIntensity2Desc := #C_ProcessLightingConfig.ColourGroupIntensity2Desc;
       #H_GBProcessLighting.H_TopCoatColourIntensity3Desc := #C_ProcessLightingConfig.ColourGroupIntensity3Desc;
   END_IF;
END_REGION

REGION Network 27: **** 8 - Outputs **** Output 1 - Break Mode
   #O_BreakMode := #BreakMode;
END_REGION

REGION Network 28: **** 8 - Outputs **** Output 2 - Intensity 1
   #O_Intensity1 := #Intensity1;
END_REGION

REGION Network 29: **** 8 - Outputs **** Output 3 - Intensity 2
   #O_Intensity2 := #Intensity2;
END_REGION

REGION Network 30: **** 8 - Outputs **** Output 4 - Intensity 3
   #O_Intensity3 := #Intensity3;
END_REGION

REGION Network 31: **** 8 - Outputs **** Global output
   IF #IO_GlobalOutput OR #BreakMode OR #Intensity1 OR #Intensity2 OR #Intensity3 THEN
       #IO_GlobalOutput := TRUE;
   END_IF;
END_REGION

REGION Network 32: **** 8 - Outputs **** Alarm AB Condition
   // Alarm AB Condition
   #O_AlarmABCondition := "FALSE" OR "FALSE";
   #AlarmABCondition := #O_AlarmABCondition;
END_REGION

REGION Network 33: **** 9 - Alarm Summary **** Alarm A
   // Alarm A
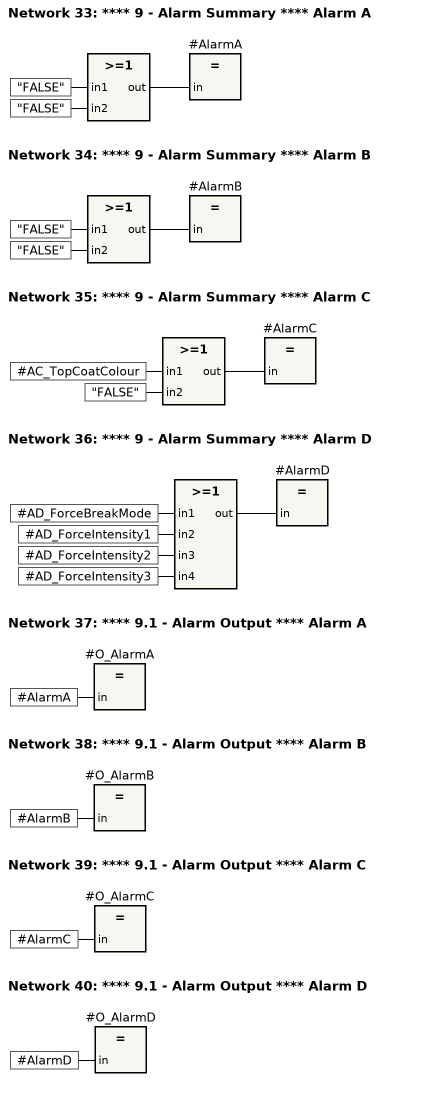
   #AlarmA := "FALSE" OR "FALSE";
END_REGION

REGION Network 34: **** 9 - Alarm Summary **** Alarm B
   // Alarm B
   #AlarmB := "FALSE" OR "FALSE";
END_REGION

REGION Network 35: **** 9 - Alarm Summary **** Alarm C
   // Alarm C
   #AlarmC := #AC_TopCoatColour OR "FALSE";
END_REGION

REGION Network 36: **** 9 - Alarm Summary **** Alarm D
   // Alarm D
   #AlarmD := #AD_ForceBreakMode OR #AD_ForceIntensity1 OR #AD_ForceIntensity2 OR #AD_ForceIntensity3;
END_REGION

REGION Network 37: **** 9.1 - Alarm Output **** Alarm A
   // Alarm A
   #O_AlarmA := #AlarmA;
END_REGION

REGION Network 38: **** 9.1 - Alarm Output **** Alarm B
   // Alarm B
   #O_AlarmB := #AlarmB;
END_REGION

REGION Network 39: **** 9.1 - Alarm Output **** Alarm C
   // Alarm C
   #O_AlarmC := #AlarmC;
END_REGION

REGION Network 40: **** 9.1 - Alarm Output **** Alarm D
   // Alarm D
   #O_AlarmD := #AlarmD;
END_REGION

REGION Network 41: **** 9.2 - Alarm DWord**** Alarm To DWord
   // Alarm To DWord
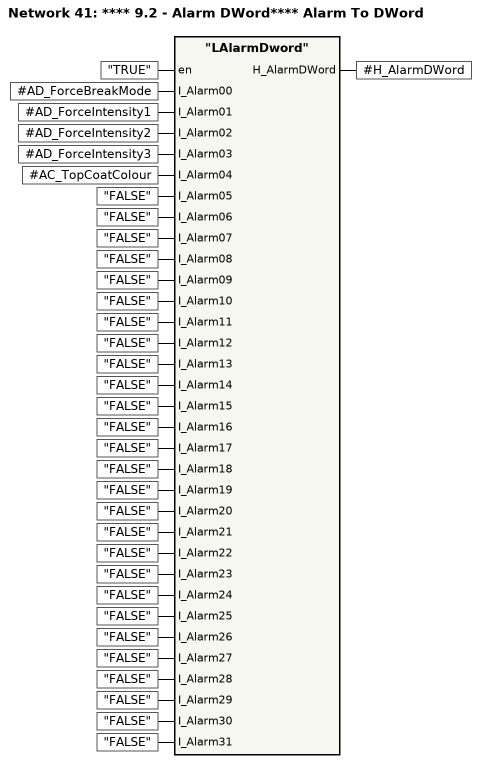
   IF "TRUE" THEN
       "LAlarmDword"(I_Alarm00 := #AD_ForceBreakMode,
                     I_Alarm01 := #AD_ForceIntensity1,
                     I_Alarm02 := #AD_ForceIntensity2,
                     I_Alarm03 := #AD_ForceIntensity3,
                     I_Alarm04 := #AC_TopCoatColour,
                     I_Alarm05 := "FALSE",
                     I_Alarm06 := "FALSE",
                     I_Alarm07 := "FALSE",
                     I_Alarm08 := "FALSE",
                     I_Alarm09 := "FALSE",
                     I_Alarm10 := "FALSE",
                     I_Alarm11 := "FALSE",
                     I_Alarm12 := "FALSE",
                     I_Alarm13 := "FALSE",
                     I_Alarm14 := "FALSE",
                     I_Alarm15 := "FALSE",
                     I_Alarm16 := "FALSE",
                     I_Alarm17 := "FALSE",
                     I_Alarm18 := "FALSE",
                     I_Alarm19 := "FALSE",
                     I_Alarm20 := "FALSE",
                     I_Alarm21 := "FALSE",
                     I_Alarm22 := "FALSE",
                     I_Alarm23 := "FALSE",
                     I_Alarm24 := "FALSE",
                     I_Alarm25 := "FALSE",
                     I_Alarm26 := "FALSE",
                     I_Alarm27 := "FALSE",
                     I_Alarm28 := "FALSE",
                     I_Alarm29 := "FALSE",
                     I_Alarm30 := "FALSE",
                     I_Alarm31 := "FALSE",
                     H_AlarmDWord => #H_AlarmDWord);
   END_IF;
END_REGION
END_FUNCTION_BLOCK
